(* PLC project PLC_NeuralNetwork, Beckhoff Automation GmbH TwinCAT PLC Control 3.5.13.21 *)
(* stored: creationDateTime 2024-04-22T16:02:21.5154165, modificationDateTime 2024-04-22T16:02:21.5174167 *)

PROGRAM MAIN
  VAR CONSTANT
    cModelInputChannels : UDINT := 3;
    cModelInputWidth : UDINT := 224;
    cModelInputHeight : UDINT := 224;
    cMaxPixelValue : UDINT := 255;
    cNumberOfClasses : UDINT := 21;
  END_VAR
  VAR
    hr : HRESULT;
    fbCameraControl : FB_VN_SimpleCameraControl;
    eCameraState : ETcVnCameraState;
    sFolderPath : STRING(255) := 'C:\cnnModels\';  (* Load Model *)
    sFilePath : STRING(255);
    fbReadDnn : FB_VN_ReadNeuralNetwork;
    ipDnnModel : ITcVnNeuralNetwork;
    bDnnModelInitialized : BOOL := FALSE;
    nReturnCode : UDINT;
    sFileName : STRING(255);  (* Model information *)
    sClassLabels : ARRAY[0..cNumberOfClasses] OF STRING := ['nok_kratzer: ', 'ok: '];
    aMean : TcVnVector4_LREAL := [0.229, 0.224, 0.225];
    aStd : TcVnVector4_LREAL := [0.485, 0.456, 0.406];
    ePaddingMode : ETcVnPaddingMode := TCVN_PM_CROP_CENTER;
    eInterpolationType : ETcVnInterpolationType := TCVN_IT_BILINEAR;
    ipImageIn : ITcVnImage;  (* Images *)
    ipImageInDisp : ITcVnDisplayableImage;
    stPixelFormat : TcVnPixelFormat;
    ipTensorImage : ITcVnImage;
    ipDnnOutputImage : ITcVnImage;
    aConfidence : TcVnVector4_LREAL;  (* Result *)
    aClassIndex : TcVnPoint2_DINT;
    sResult : STRING(255);
    aWhite : TcVnVector4_LREAL := [255, 255, 255];
    aBlack : TcVnVector4_LREAL := [0, 0, 0];
  END_VAR

            // Disclaimer

// This publication contains statements about the suitability of our products for certain
// areas of application. These statements are based on typical features of our products.
// The examples shown in this publication are for demonstration purposes only.
// The information provided herein should not be regarded as specific operation characteristics.
// It is incumbent on the customer to check and decide whether a product is suitable for use
// in a particular application. We do not give any warranty that the source code which is
// made available with this publication is complete or accurate.

// THE SAMPLE CODE CONTAINED IN THIS PUBLICATION IS PROVIDED “AS IS” WITHOUT WARRANTY OF ANY KIND,
// EITHER EXPRESSED, IMPLIED OR STATUTORY, INCLUDING WITHOUT LIMITATION, ANY WARRANTY WITH RESPECT TO NON-INFRINGEMENT,
// FREEDOM FROM PROPRIETARY RIGHTS OF THIRD PARTIES OR FITNESS FOR ANY PARTICULAR PURPOSE.

// This publication may be changed from time to time without prior notice.
// No liability is assumed for errors and/or omissions.
// Our products are described in detail in our data sheets and documentations.
// Product-specific warnings and cautions must be observed.
// For the latest version of our data sheets and documentations visit our website (www.beckhoff.de).

// © Beckhoff Automation GmbH & Co. KG, December 2023

// The reproduction, distribution and utilization of this document as well as the communication
// of its contents to others without express authorization is prohibited.
// Offenders will be held liable for the payment of damages.
// All rights reserved in the event of the grant of a patent, utility model or design.

//	==========================================================================================

// SAMPLE - Neural Network
//	-------------------------------------------------------

// Steps To Do:
// ------------
// 1. Add the images to the FileSource control
// 2. Activate the configuration -> Start TwinCAT system and PLC to run
// 3. Watch the results in the ADS Image Watch

// Load Dnn model
IF NOT bDnnModelInitialized THEN
	sFilePath := CONCAT (sFolderPath,sFileName);
	FW_SafeRelease(ADR(ipDnnModel));
	fbReadDnn(sFilePath := sFilePath, ipDestNeuralNetwork := ipDnnModel, bRead := TRUE);

	IF NOT fbReadDnn.bBusy THEN
		fbReadDnn(sFilePath:='', bRead := FALSE);
		IF NOT fbReadDnn.bError THEN
			bDnnModelInitialized := TRUE;
		END_IF
		nReturnCode := fbReadDnn.nErrorId AND 16#FFF;
	END_IF
END_IF

// Get camera state
eCameraState := fbCameraControl.GetState();

// CameraControl is in error state
IF eCameraState = TCVN_CS_ERROR THEN
	hr := fbCameraControl.Reset();

// Camera not yet streaming
ELSIF eCameraState < TCVN_CS_ACQUIRING THEN
	hr := fbCameraControl.StartAcquisition();

// Camera streaming
ELSIF eCameraState = TCVN_CS_ACQUIRING THEN
	hr := fbCameraControl.GetCurrentImage(ipImageIn);

	// Check if new image was received
	IF bDnnModelInitialized AND SUCCEEDED(hr) AND ipImageIn <> 0 THEN
		hr := F_VN_GetPixelFormat(ipImageIn, stPixelFormat, hr);

		// Check if input image channels matches the model requirements, alternative implement the needed color space transformation yourself.
		IF stPixelFormat.nChannels <> cModelInputChannels OR stPixelFormat.ePixelEncoding <> TCVN_PE_NONE THEN
			hr := Tc2_System.E_HRESULTAdsErr.INCOMPATIBLE;
		END_IF

		// *** Preprocessing steps ***
		// Adjust the dimensions of the input image to match the model input requirements
		hr := F_VN_ResizeImageExp(ipImageIn, ipTensorImage, cModelInputWidth, cModelInputHeight, eInterpolationType, ePaddingMode, aBlack, hr);

		// Convert the image to type REAL and scale to the range [0.0, 1.0]
		hr := F_VN_ConvertElementTypeExp(ipTensorImage, ipTensorImage, TCVN_ET_REAL, 1.0 / UDINT_TO_REAL(cMaxPixelValue), 0, hr);

		// Normalization
		hr := F_VN_SubtractVectorFromImage(ipTensorImage, aMean, ipTensorImage,hr);
		hr := F_VN_DivideImageByVector(ipTensorImage, aStd, ipTensorImage, hr);

		// Convert the input image to 4D Tensor
		hr := F_VN_ConvertDataLayout(ipTensorImage, ipTensorImage, TCVN_DL_4D_NCHW, hr);

		// *** Model execution ***
		hr := F_VN_ExecuteNeuralNetwork(ipDnnModel, ipTensorImage, ipDnnOutputImage, hr);

		// *** Postprocessing steps ***
		// Get best classfication result
		hr := F_VN_SoftMax(ipDnnOutputImage,ipDnnOutputImage,hr);
		hr := F_VN_MaxPixelValue(ipDnnOutputImage, aConfidence , aClassIndex, hr);

		// Result visualization
		sResult := CONCAT(sClassLabels[aClassIndex[0]] , LREAL_TO_FMTSTR(aConfidence[0], 2, FALSE));
		hr := F_VN_PutLabelExp(sResult, ipImageIn, 5, 15, 1, 1, TCVN_FT_HERSHEY_PLAIN, aBlack, aWhite, TCVN_LT_4_CONNECTED, hr);

		// Display images and release pointer
		hr := F_VN_TransformIntoDisplayableImage(ipImageIn, ipImageInDisp, S_OK);
		FW_SafeRelease(ADR(ipTensorImage));
		FW_SafeRelease(ADR(ipDnnOutputImage));
    END_IF
END_IF

          
END_PROGRAM
